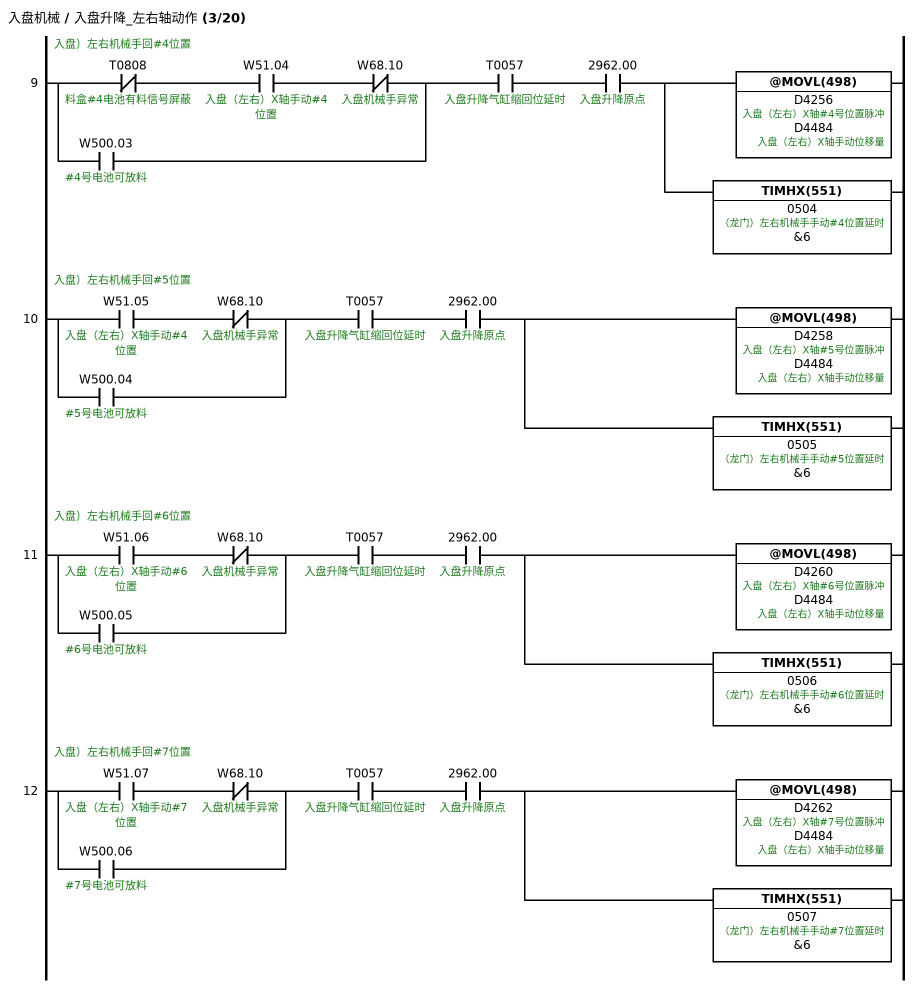
; [picture p192: 入盘机械 / 入盘升降_左右轴动作, rungs 9-12]
; rung 9: 入盘）左右机械手回#4位置
LDNOT T0808  ; 料盒#4电池有料信号屏蔽
AND W51.04  ; 入盘（左右）X轴手动#4位置
ANDNOT W68.10  ; 入盘机械手异常
OR W500.03  ; #4号电池可放料
AND T0057  ; 入盘升降气缸缩回位延时
AND 2962.00  ; 入盘升降原点
@MOVL(498) D4256 D4484  ; 入盘（左右）X轴#4号位置脉冲, 入盘（左右）X轴手动位移量
TIMHX(551) 0504 &6  ; （龙门）左右机械手手动#4位置延时
; rung 10: 入盘）左右机械手回#5位置
LD W51.05  ; 入盘（左右）X轴手动#4位置
ANDNOT W68.10  ; 入盘机械手异常
OR W500.04  ; #5号电池可放料
AND T0057  ; 入盘升降气缸缩回位延时
AND 2962.00  ; 入盘升降原点
@MOVL(498) D4258 D4484  ; 入盘（左右）X轴#5号位置脉冲, 入盘（左右）X轴手动位移量
TIMHX(551) 0505 &6  ; （龙门）左右机械手手动#5位置延时
; rung 11: 入盘）左右机械手回#6位置
LD W51.06  ; 入盘（左右）X轴手动#6位置
ANDNOT W68.10  ; 入盘机械手异常
OR W500.05  ; #6号电池可放料
AND T0057  ; 入盘升降气缸缩回位延时
AND 2962.00  ; 入盘升降原点
@MOVL(498) D4260 D4484  ; 入盘（左右）X轴#6号位置脉冲, 入盘（左右）X轴手动位移量
TIMHX(551) 0506 &6  ; （龙门）左右机械手手动#6位置延时
; rung 12: 入盘）左右机械手回#7位置
LD W51.07  ; 入盘（左右）X轴手动#7位置
ANDNOT W68.10  ; 入盘机械手异常
OR W500.06  ; #7号电池可放料
AND T0057  ; 入盘升降气缸缩回位延时
AND 2962.00  ; 入盘升降原点
@MOVL(498) D4262 D4484  ; 入盘（左右）X轴#7号位置脉冲, 入盘（左右）X轴手动位移量
TIMHX(551) 0507 &6  ; （龙门）左右机械手手动#7位置延时

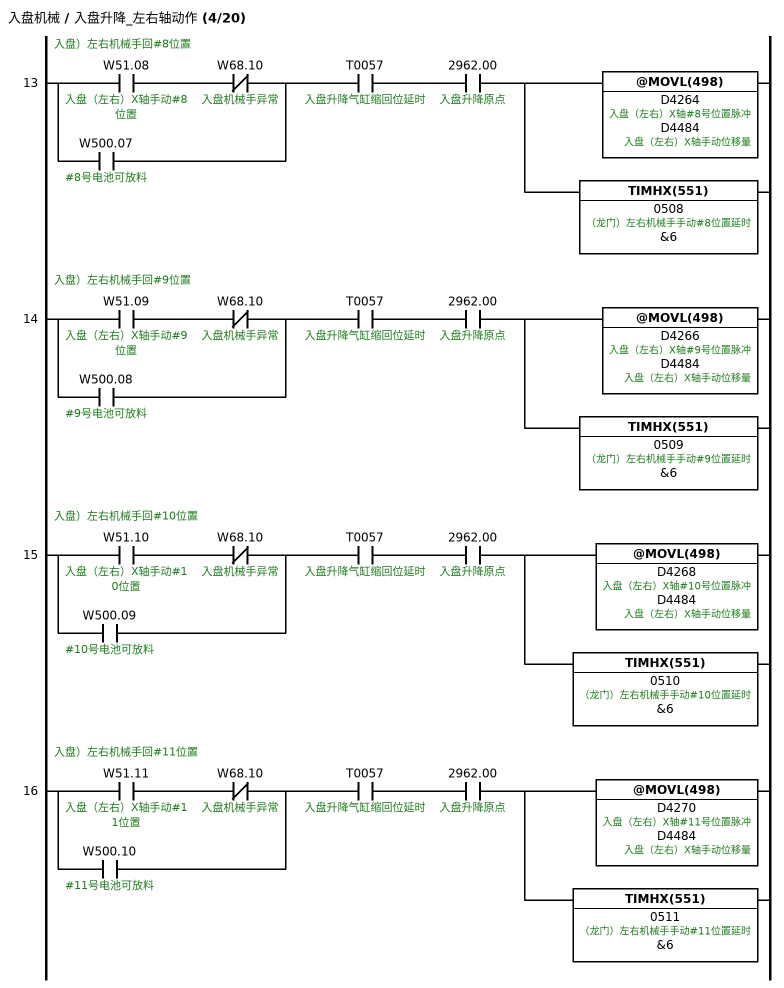
; rung 13: 入盘）左右机械手回#8位置
LD W51.08  ; 入盘（左右）X轴手动#8位置
ANDNOT W68.10  ; 入盘机械手异常
OR W500.07  ; #8号电池可放料
AND T0057  ; 入盘升降气缸缩回位延时
AND 2962.00  ; 入盘升降原点
@MOVL(498) D4264 D4484  ; 入盘（左右）X轴#8号位置脉冲, 入盘（左右）X轴手动位移量
TIMHX(551) 0508 &6  ; （龙门）左右机械手手动#8位置延时
; rung 14: 入盘）左右机械手回#9位置
LD W51.09  ; 入盘（左右）X轴手动#9位置
ANDNOT W68.10  ; 入盘机械手异常
OR W500.08  ; #9号电池可放料
AND T0057  ; 入盘升降气缸缩回位延时
AND 2962.00  ; 入盘升降原点
@MOVL(498) D4266 D4484  ; 入盘（左右）X轴#9号位置脉冲, 入盘（左右）X轴手动位移量
TIMHX(551) 0509 &6  ; （龙门）左右机械手手动#9位置延时
; rung 15: 入盘）左右机械手回#10位置
LD W51.10  ; 入盘（左右）X轴手动#10位置
ANDNOT W68.10  ; 入盘机械手异常
OR W500.09  ; #10号电池可放料
AND T0057  ; 入盘升降气缸缩回位延时
AND 2962.00  ; 入盘升降原点
@MOVL(498) D4268 D4484  ; 入盘（左右）X轴#10号位置脉冲, 入盘（左右）X轴手动位移量
TIMHX(551) 0510 &6  ; （龙门）左右机械手手动#10位置延时
; rung 16: 入盘）左右机械手回#11位置
LD W51.11  ; 入盘（左右）X轴手动#11位置
ANDNOT W68.10  ; 入盘机械手异常
OR W500.10  ; #11号电池可放料
AND T0057  ; 入盘升降气缸缩回位延时
AND 2962.00  ; 入盘升降原点
@MOVL(498) D4270 D4484  ; 入盘（左右）X轴#11号位置脉冲, 入盘（左右）X轴手动位移量
TIMHX(551) 0511 &6  ; （龙门）左右机械手手动#11位置延时

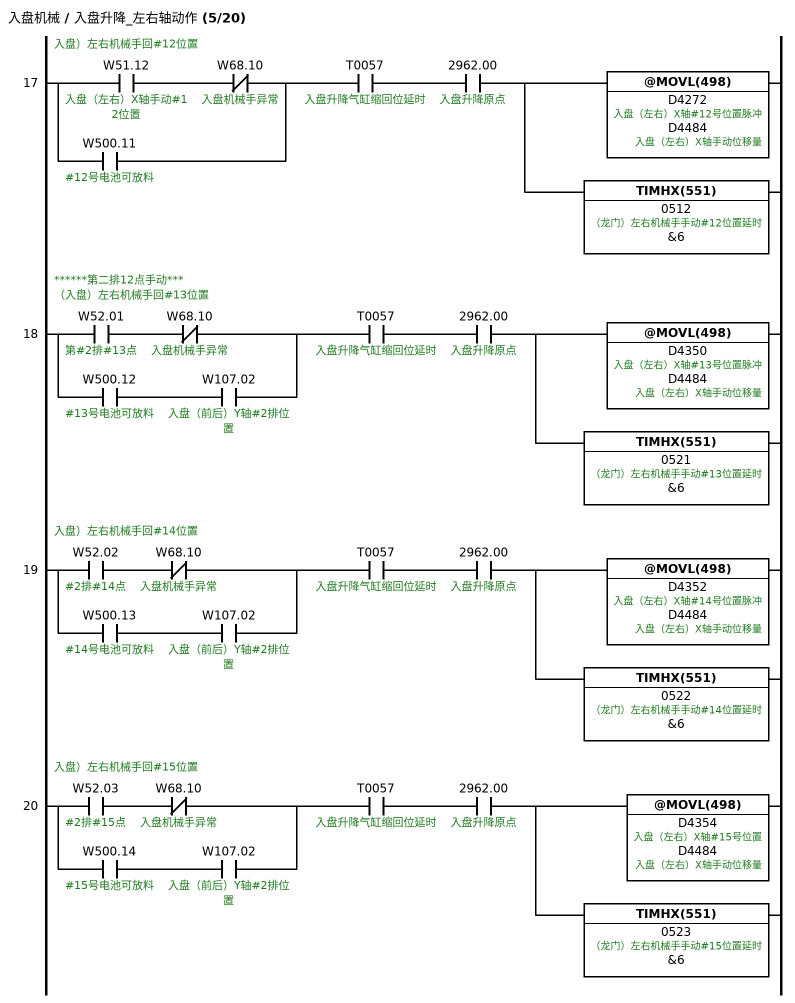
; rung 17: 入盘）左右机械手回#12位置
LD W51.12  ; 入盘（左右）X轴手动#12位置
ANDNOT W68.10  ; 入盘机械手异常
OR W500.11  ; #12号电池可放料
AND T0057  ; 入盘升降气缸缩回位延时
AND 2962.00  ; 入盘升降原点
@MOVL(498) D4272 D4484  ; 入盘（左右）X轴#12号位置脉冲, 入盘（左右）X轴手动位移量
TIMHX(551) 0512 &6  ; （龙门）左右机械手手动#12位置延时
; rung 18: ******第二排12点手动*** / （入盘）左右机械手回#13位置
LD W52.01  ; 第#2排#13点
ANDNOT W68.10  ; 入盘机械手异常
LD W500.12  ; #13号电池可放料
AND W107.02  ; 入盘（前后）Y轴#2排位置
ORLD
AND T0057  ; 入盘升降气缸缩回位延时
AND 2962.00  ; 入盘升降原点
@MOVL(498) D4350 D4484  ; 入盘（左右）X轴#13号位置脉冲, 入盘（左右）X轴手动位移量
TIMHX(551) 0521 &6  ; （龙门）左右机械手手动#13位置延时
; rung 19: 入盘）左右机械手回#14位置
LD W52.02  ; #2排#14点
ANDNOT W68.10  ; 入盘机械手异常
LD W500.13  ; #14号电池可放料
AND W107.02  ; 入盘（前后）Y轴#2排位置
ORLD
AND T0057  ; 入盘升降气缸缩回位延时
AND 2962.00  ; 入盘升降原点
@MOVL(498) D4352 D4484  ; 入盘（左右）X轴#14号位置脉冲, 入盘（左右）X轴手动位移量
TIMHX(551) 0522 &6  ; （龙门）左右机械手手动#14位置延时
; rung 20: 入盘）左右机械手回#15位置
LD W52.03  ; #2排#15点
ANDNOT W68.10  ; 入盘机械手异常
LD W500.14  ; #15号电池可放料
AND W107.02  ; 入盘（前后）Y轴#2排位置
ORLD
AND T0057  ; 入盘升降气缸缩回位延时
AND 2962.00  ; 入盘升降原点
@MOVL(498) D4354 D4484  ; 入盘（左右）X轴#15号位置, 入盘（左右）X轴手动位移量
TIMHX(551) 0523 &6  ; （龙门）左右机械手手动#15位置延时

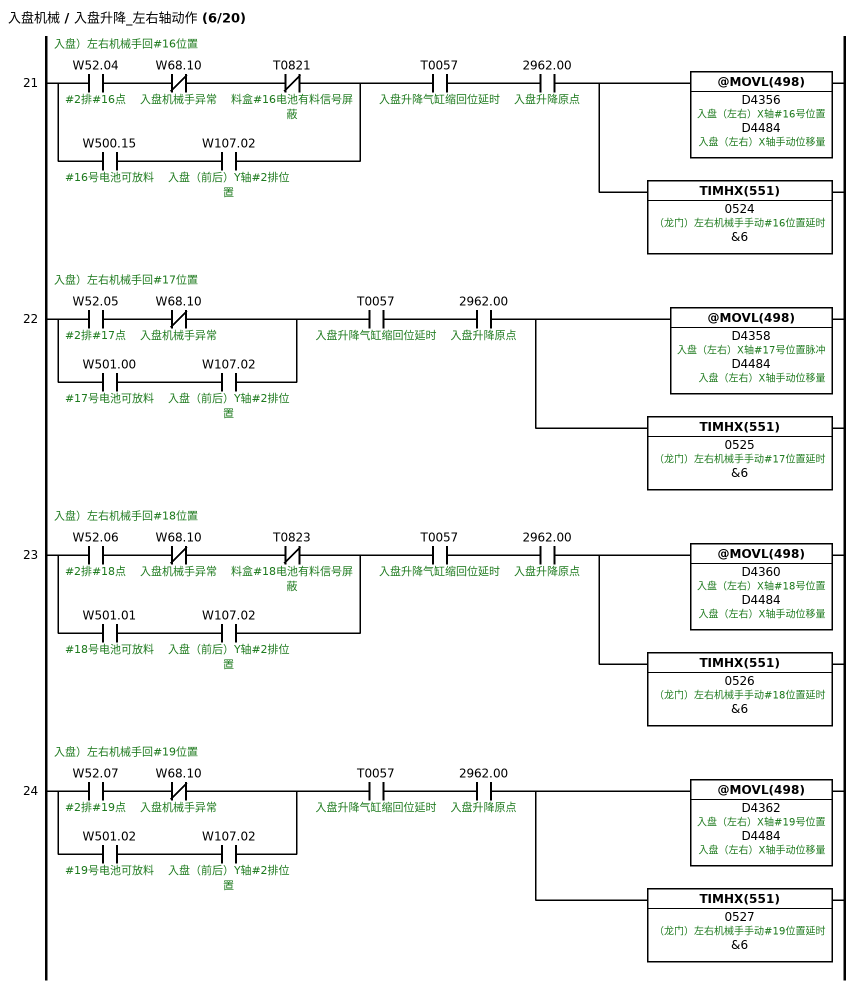
; rung 21: 入盘）左右机械手回#16位置
LD W52.04  ; #2排#16点
ANDNOT W68.10  ; 入盘机械手异常
ANDNOT T0821  ; 料盒#16电池有料信号屏蔽
LD W500.15  ; #16号电池可放料
AND W107.02  ; 入盘（前后）Y轴#2排位置
ORLD
AND T0057  ; 入盘升降气缸缩回位延时
AND 2962.00  ; 入盘升降原点
@MOVL(498) D4356 D4484  ; 入盘（左右）X轴#16号位置, 入盘（左右）X轴手动位移量
TIMHX(551) 0524 &6  ; （龙门）左右机械手手动#16位置延时
; rung 22: 入盘）左右机械手回#17位置
LD W52.05  ; #2排#17点
ANDNOT W68.10  ; 入盘机械手异常
LD W501.00  ; #17号电池可放料
AND W107.02  ; 入盘（前后）Y轴#2排位置
ORLD
AND T0057  ; 入盘升降气缸缩回位延时
AND 2962.00  ; 入盘升降原点
@MOVL(498) D4358 D4484  ; 入盘（左右）X轴#17号位置脉冲, 入盘（左右）X轴手动位移量
TIMHX(551) 0525 &6  ; （龙门）左右机械手手动#17位置延时
; rung 23: 入盘）左右机械手回#18位置
LD W52.06  ; #2排#18点
ANDNOT W68.10  ; 入盘机械手异常
ANDNOT T0823  ; 料盒#18电池有料信号屏蔽
LD W501.01  ; #18号电池可放料
AND W107.02  ; 入盘（前后）Y轴#2排位置
ORLD
AND T0057  ; 入盘升降气缸缩回位延时
AND 2962.00  ; 入盘升降原点
@MOVL(498) D4360 D4484  ; 入盘（左右）X轴#18号位置, 入盘（左右）X轴手动位移量
TIMHX(551) 0526 &6  ; （龙门）左右机械手手动#18位置延时
; rung 24: 入盘）左右机械手回#19位置
LD W52.07  ; #2排#19点
ANDNOT W68.10  ; 入盘机械手异常
LD W501.02  ; #19号电池可放料
AND W107.02  ; 入盘（前后）Y轴#2排位置
ORLD
AND T0057  ; 入盘升降气缸缩回位延时
AND 2962.00  ; 入盘升降原点
@MOVL(498) D4362 D4484  ; 入盘（左右）X轴#19号位置, 入盘（左右）X轴手动位移量
TIMHX(551) 0527 &6  ; （龙门）左右机械手手动#19位置延时

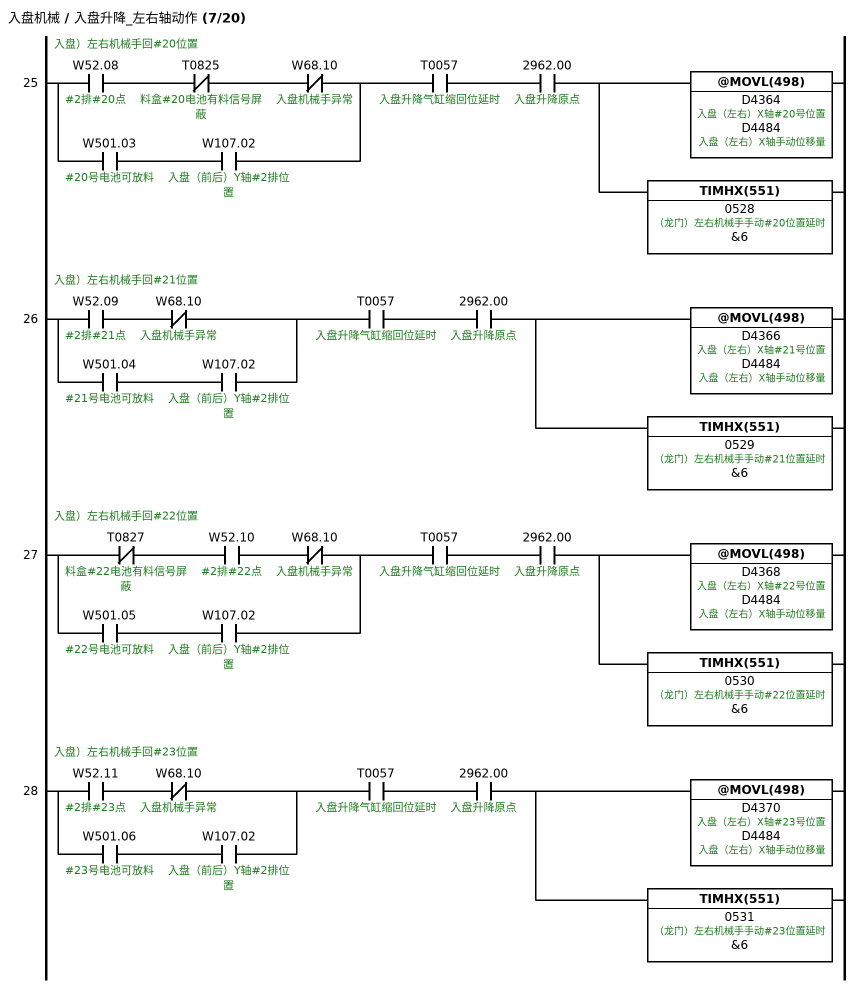
; rung 25: 入盘）左右机械手回#20位置
LD W52.08  ; #2排#20点
ANDNOT T0825  ; 料盒#20电池有料信号屏蔽
ANDNOT W68.10  ; 入盘机械手异常
LD W501.03  ; #20号电池可放料
AND W107.02  ; 入盘（前后）Y轴#2排位置
ORLD
AND T0057  ; 入盘升降气缸缩回位延时
AND 2962.00  ; 入盘升降原点
@MOVL(498) D4364 D4484  ; 入盘（左右）X轴#20号位置, 入盘（左右）X轴手动位移量
TIMHX(551) 0528 &6  ; （龙门）左右机械手手动#20位置延时
; rung 26: 入盘）左右机械手回#21位置
LD W52.09  ; #2排#21点
ANDNOT W68.10  ; 入盘机械手异常
LD W501.04  ; #21号电池可放料
AND W107.02  ; 入盘（前后）Y轴#2排位置
ORLD
AND T0057  ; 入盘升降气缸缩回位延时
AND 2962.00  ; 入盘升降原点
@MOVL(498) D4366 D4484  ; 入盘（左右）X轴#21号位置, 入盘（左右）X轴手动位移量
TIMHX(551) 0529 &6  ; （龙门）左右机械手手动#21位置延时
; rung 27: 入盘）左右机械手回#22位置
LDNOT T0827  ; 料盒#22电池有料信号屏蔽
AND W52.10  ; #2排#22点
ANDNOT W68.10  ; 入盘机械手异常
LD W501.05  ; #22号电池可放料
AND W107.02  ; 入盘（前后）Y轴#2排位置
ORLD
AND T0057  ; 入盘升降气缸缩回位延时
AND 2962.00  ; 入盘升降原点
@MOVL(498) D4368 D4484  ; 入盘（左右）X轴#22号位置, 入盘（左右）X轴手动位移量
TIMHX(551) 0530 &6  ; （龙门）左右机械手手动#22位置延时
; rung 28: 入盘）左右机械手回#23位置
LD W52.11  ; #2排#23点
ANDNOT W68.10  ; 入盘机械手异常
LD W501.06  ; #23号电池可放料
AND W107.02  ; 入盘（前后）Y轴#2排位置
ORLD
AND T0057  ; 入盘升降气缸缩回位延时
AND 2962.00  ; 入盘升降原点
@MOVL(498) D4370 D4484  ; 入盘（左右）X轴#23号位置, 入盘（左右）X轴手动位移量
TIMHX(551) 0531 &6  ; （龙门）左右机械手手动#23位置延时

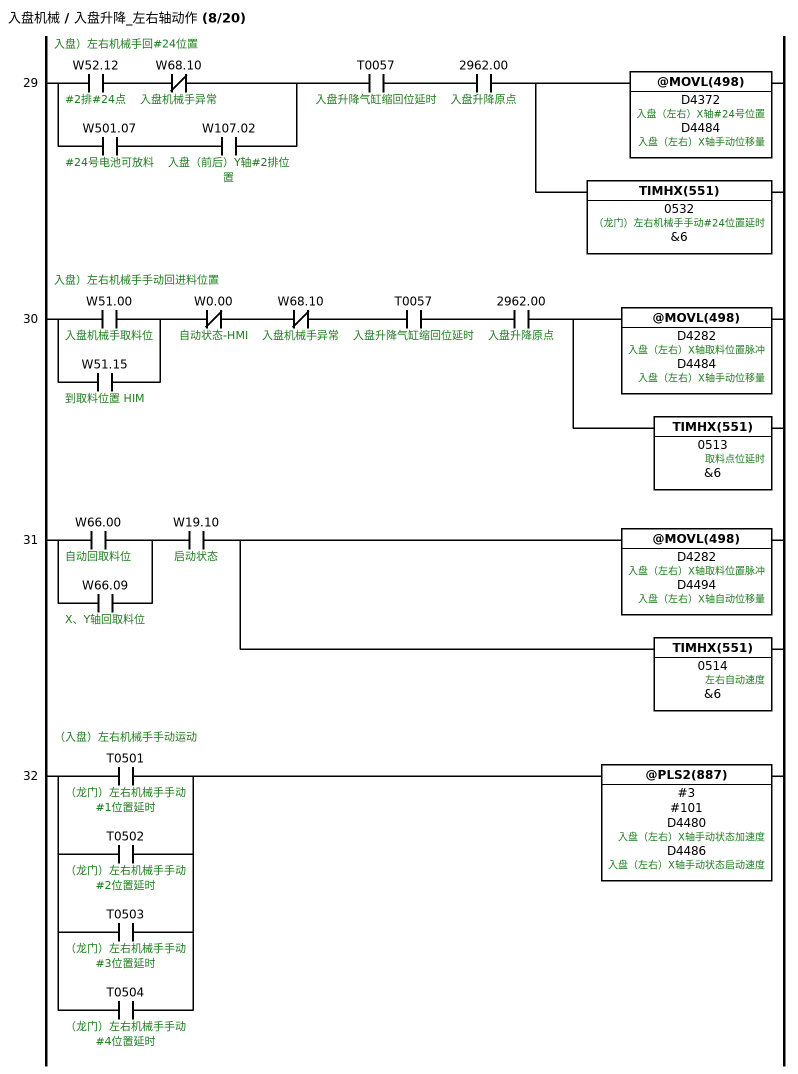
; rung 29: 入盘）左右机械手回#24位置
LD W52.12  ; #2排#24点
ANDNOT W68.10  ; 入盘机械手异常
LD W501.07  ; #24号电池可放料
AND W107.02  ; 入盘（前后）Y轴#2排位置
ORLD
AND T0057  ; 入盘升降气缸缩回位延时
AND 2962.00  ; 入盘升降原点
@MOVL(498) D4372 D4484  ; 入盘（左右）X轴#24号位置, 入盘（左右）X轴手动位移量
TIMHX(551) 0532 &6  ; （龙门）左右机械手手动#24位置延时
; rung 30: 入盘）左右机械手手动回进料位置
LD W51.00  ; 入盘机械手取料位
OR W51.15  ; 到取料位置 HIM
ANDNOT W0.00  ; 自动状态-HMI
ANDNOT W68.10  ; 入盘机械手异常
AND T0057  ; 入盘升降气缸缩回位延时
AND 2962.00  ; 入盘升降原点
@MOVL(498) D4282 D4484  ; 入盘（左右）X轴取料位置脉冲, 入盘（左右）X轴手动位移量
TIMHX(551) 0513 &6  ; 取料点位延时
; rung 31
LD W66.00  ; 自动回取料位
OR W66.09  ; X、Y轴回取料位
AND W19.10  ; 启动状态
@MOVL(498) D4282 D4494  ; 入盘（左右）X轴取料位置脉冲, 入盘（左右）X轴自动位移量
TIMHX(551) 0514 &6  ; 左右自动速度
; rung 32: （入盘）左右机械手手动运动
LD T0501  ; （龙门）左右机械手手动#1位置延时
OR T0502  ; （龙门）左右机械手手动#2位置延时
OR T0503  ; （龙门）左右机械手手动#3位置延时
OR T0504  ; （龙门）左右机械手手动#4位置延时
@PLS2(887) #3 #101 D4480 D4486  ; 入盘（左右）X轴手动状态加速度, 入盘（左右）X轴手动状态启动速度

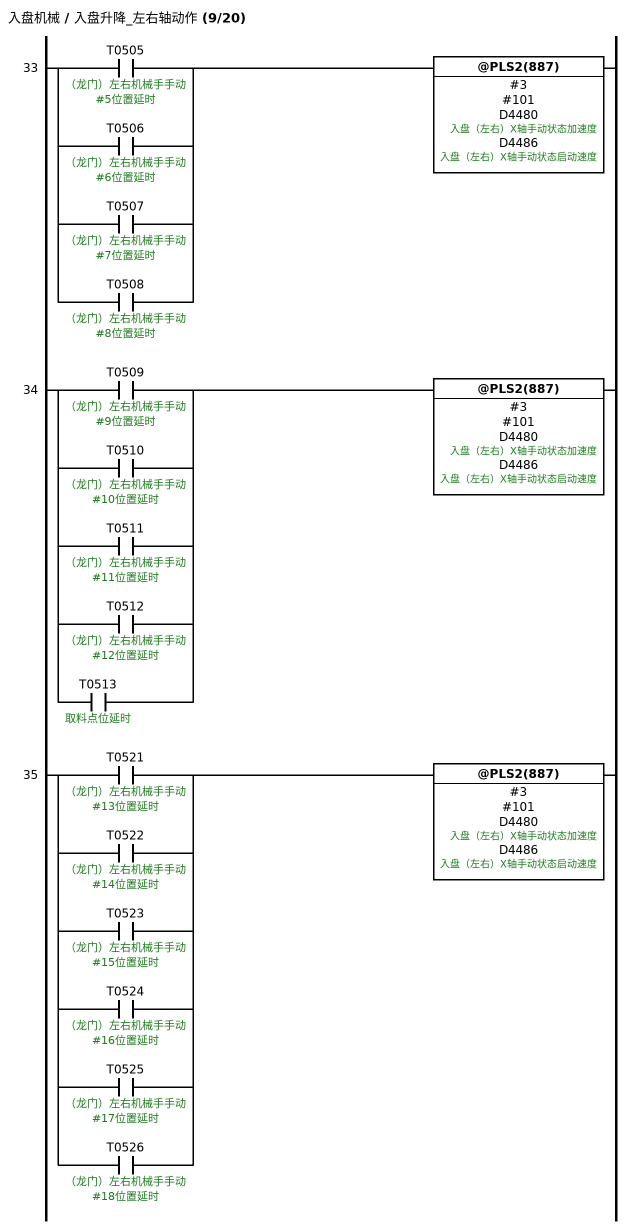
; rung 33
LD T0505  ; （龙门）左右机械手手动#5位置延时
OR T0506  ; （龙门）左右机械手手动#6位置延时
OR T0507  ; （龙门）左右机械手手动#7位置延时
OR T0508  ; （龙门）左右机械手手动#8位置延时
@PLS2(887) #3 #101 D4480 D4486  ; 入盘（左右）X轴手动状态加速度, 入盘（左右）X轴手动状态启动速度
; rung 34
LD T0509  ; （龙门）左右机械手手动#9位置延时
OR T0510  ; （龙门）左右机械手手动#10位置延时
OR T0511  ; （龙门）左右机械手手动#11位置延时
OR T0512  ; （龙门）左右机械手手动#12位置延时
OR T0513  ; 取料点位延时
@PLS2(887) #3 #101 D4480 D4486  ; 入盘（左右）X轴手动状态加速度, 入盘（左右）X轴手动状态启动速度
; rung 35
LD T0521  ; （龙门）左右机械手手动#13位置延时
OR T0522  ; （龙门）左右机械手手动#14位置延时
OR T0523  ; （龙门）左右机械手手动#15位置延时
OR T0524  ; （龙门）左右机械手手动#16位置延时
OR T0525  ; （龙门）左右机械手手动#17位置延时
OR T0526  ; （龙门）左右机械手手动#18位置延时
@PLS2(887) #3 #101 D4480 D4486  ; 入盘（左右）X轴手动状态加速度, 入盘（左右）X轴手动状态启动速度

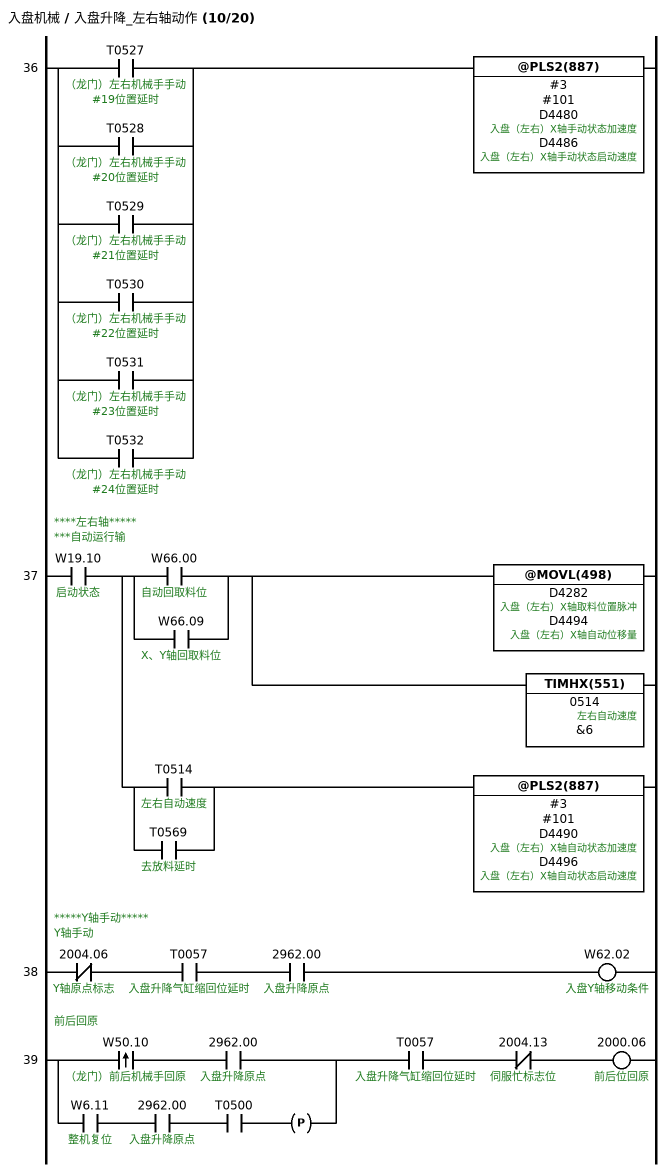
; rung 36
LD T0527  ; （龙门）左右机械手手动#19位置延时
OR T0528  ; （龙门）左右机械手手动#20位置延时
OR T0529  ; （龙门）左右机械手手动#21位置延时
OR T0530  ; （龙门）左右机械手手动#22位置延时
OR T0531  ; （龙门）左右机械手手动#23位置延时
OR T0532  ; （龙门）左右机械手手动#24位置延时
@PLS2(887) #3 #101 D4480 D4486  ; 入盘（左右）X轴手动状态加速度, 入盘（左右）X轴手动状态启动速度
; rung 37: ****左右轴***** / ***自动运行输
LD W19.10  ; 启动状态
OUT TR0
LD W66.00  ; 自动回取料位
OR W66.09  ; X、Y轴回取料位
ANDLD
@MOVL(498) D4282 D4494  ; 入盘（左右）X轴取料位置脉冲, 入盘（左右）X轴自动位移量
TIMHX(551) 0514 &6  ; 左右自动速度
LD TR0
LD T0514  ; 左右自动速度
OR T0569  ; 去放料延时
ANDLD
@PLS2(887) #3 #101 D4490 D4496  ; 入盘（左右）X轴自动状态加速度, 入盘（左右）X轴自动状态启动速度
; rung 38: *****Y轴手动***** / Y轴手动
LDNOT 2004.06  ; Y轴原点标志
AND T0057  ; 入盘升降气缸缩回位延时
AND 2962.00  ; 入盘升降原点
OUT W62.02  ; 入盘Y轴移动条件
; rung 39: 前后回原
@LD W50.10  ; （龙门）前后机械手回原
AND 2962.00  ; 入盘升降原点
LD W6.11  ; 整机复位
AND 2962.00  ; 入盘升降原点
AND T0500
UP(521)
ORLD
AND T0057  ; 入盘升降气缸缩回位延时
ANDNOT 2004.13  ; 伺服忙标志位
OUT 2000.06  ; 前后位回原

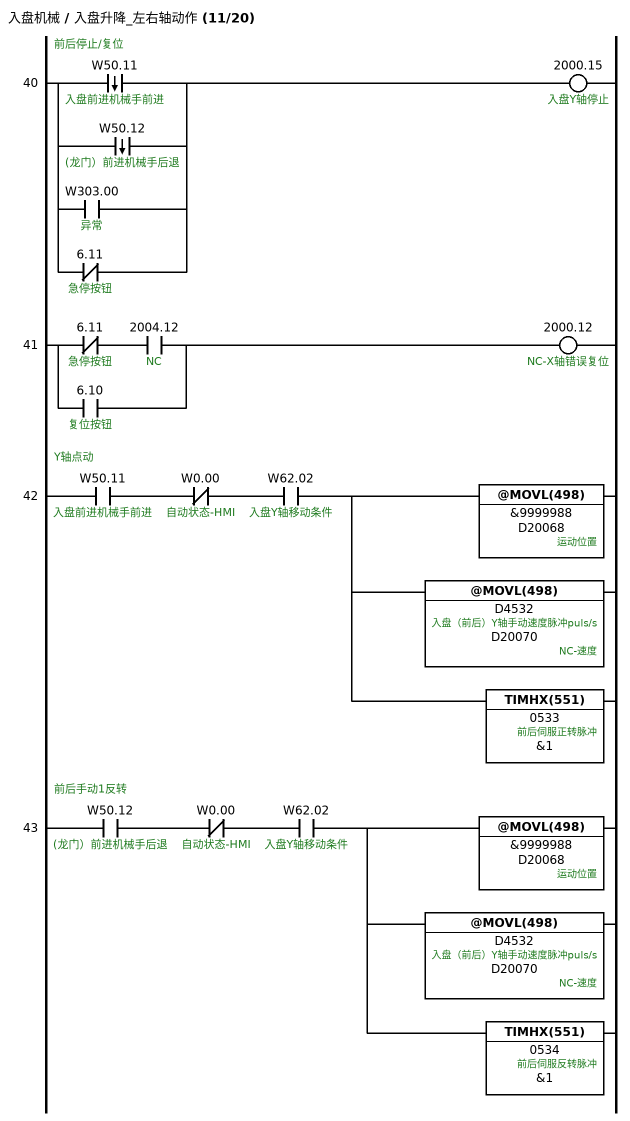
; rung 40: 前后停止/复位
%LD W50.11  ; 入盘前进机械手前进
%OR W50.12  ; (龙门）前进机械手后退
OR W303.00  ; 异常
ORNOT 6.11  ; 急停按钮
OUT 2000.15  ; 入盘Y轴停止
; rung 41
LDNOT 6.11  ; 急停按钮
AND 2004.12  ; NC
OR 6.10  ; 复位按钮
OUT 2000.12  ; NC-X轴错误复位
; rung 42: Y轴点动
LD W50.11  ; 入盘前进机械手前进
ANDNOT W0.00  ; 自动状态-HMI
AND W62.02  ; 入盘Y轴移动条件
@MOVL(498) &9999988 D20068  ; 运动位置
@MOVL(498) D4532 D20070  ; 入盘（前后）Y轴手动速度脉冲puls/s, NC-速度
TIMHX(551) 0533 &1  ; 前后伺服正转脉冲
; rung 43: 前后手动1反转
LD W50.12  ; (龙门）前进机械手后退
ANDNOT W0.00  ; 自动状态-HMI
AND W62.02  ; 入盘Y轴移动条件
@MOVL(498) &9999988 D20068  ; 运动位置
@MOVL(498) D4532 D20070  ; 入盘（前后）Y轴手动速度脉冲puls/s, NC-速度
TIMHX(551) 0534 &1  ; 前后伺服反转脉冲

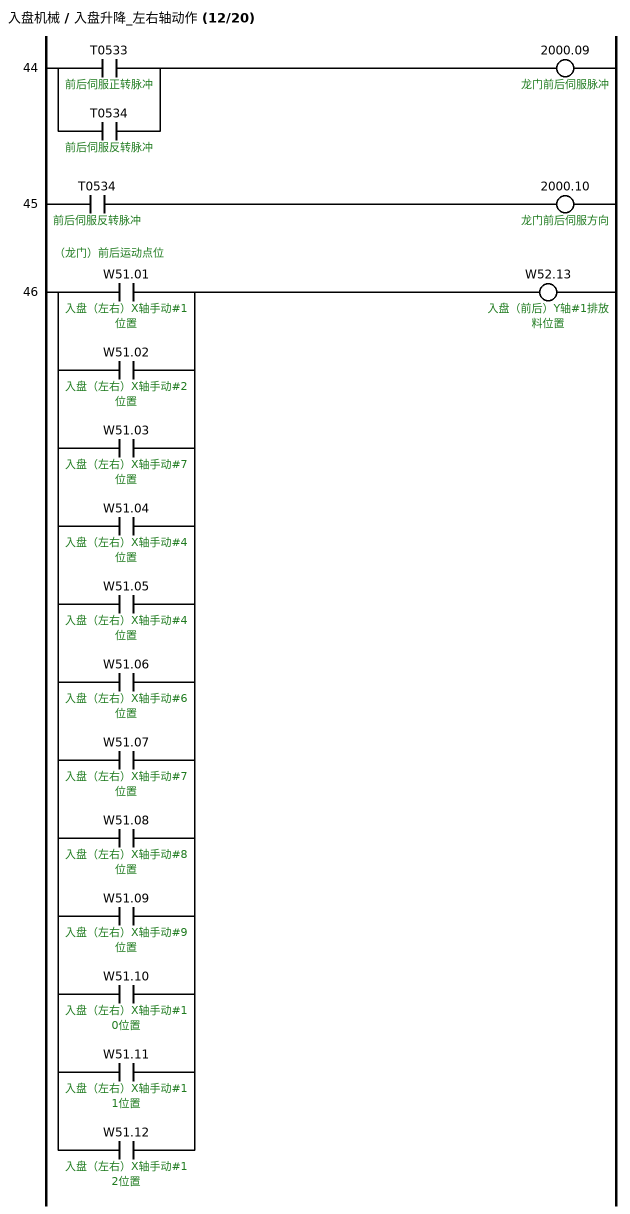
; rung 44
LD T0533  ; 前后伺服正转脉冲
OR T0534  ; 前后伺服反转脉冲
OUT 2000.09  ; 龙门前后伺服脉冲
; rung 45
LD T0534  ; 前后伺服反转脉冲
OUT 2000.10  ; 龙门前后伺服方向
; rung 46: （龙门）前后运动点位
LD W51.01  ; 入盘（左右）X轴手动#1位置
OR W51.02  ; 入盘（左右）X轴手动#2位置
OR W51.03  ; 入盘（左右）X轴手动#7位置
OR W51.04  ; 入盘（左右）X轴手动#4位置
OR W51.05  ; 入盘（左右）X轴手动#4位置
OR W51.06  ; 入盘（左右）X轴手动#6位置
OR W51.07  ; 入盘（左右）X轴手动#7位置
OR W51.08  ; 入盘（左右）X轴手动#8位置
OR W51.09  ; 入盘（左右）X轴手动#9位置
OR W51.10  ; 入盘（左右）X轴手动#10位置
OR W51.11  ; 入盘（左右）X轴手动#11位置
OR W51.12  ; 入盘（左右）X轴手动#12位置
OUT W52.13  ; 入盘（前后）Y轴#1排放料位置

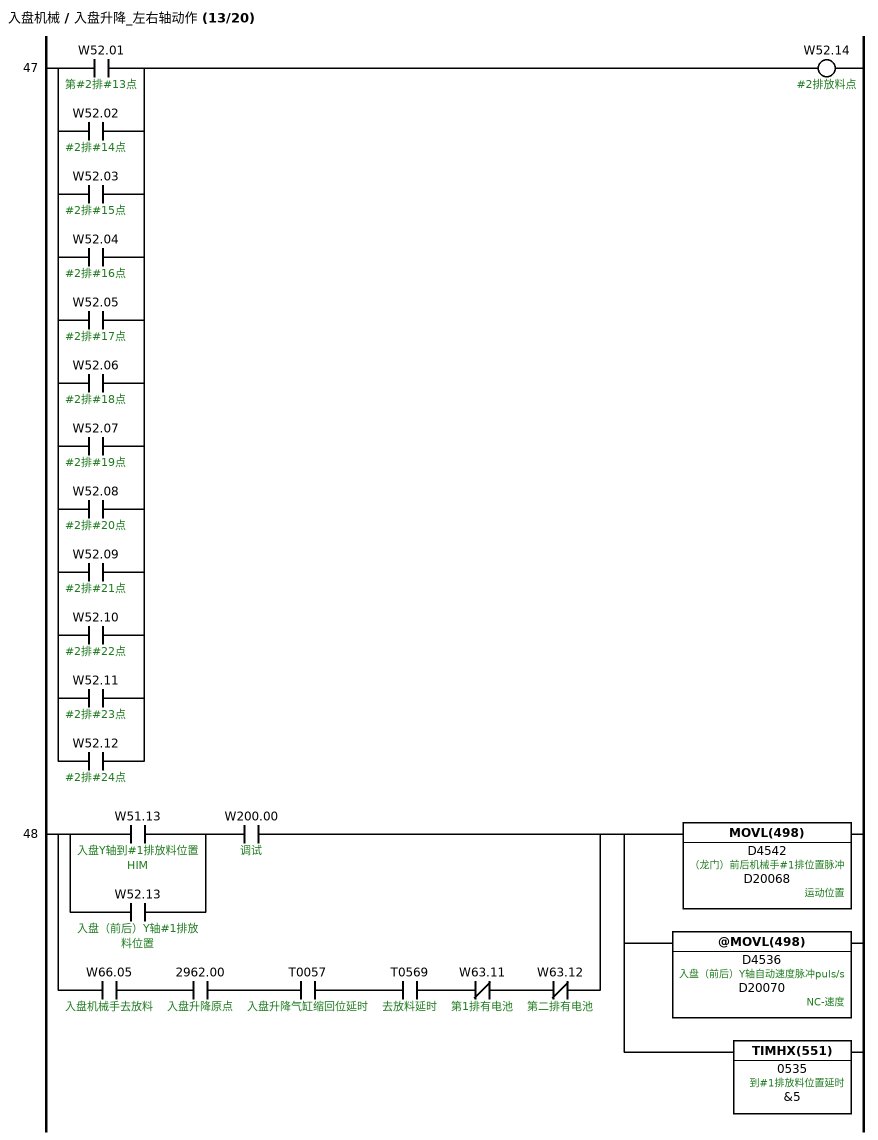
; rung 47
LD W52.01  ; 第#2排#13点
OR W52.02  ; #2排#14点
OR W52.03  ; #2排#15点
OR W52.04  ; #2排#16点
OR W52.05  ; #2排#17点
OR W52.06  ; #2排#18点
OR W52.07  ; #2排#19点
OR W52.08  ; #2排#20点
OR W52.09  ; #2排#21点
OR W52.10  ; #2排#22点
OR W52.11  ; #2排#23点
OR W52.12  ; #2排#24点
OUT W52.14  ; #2排放料点
; rung 48
LD W51.13  ; 入盘Y轴到#1排放料位置  HIM
OR W52.13  ; 入盘（前后）Y轴#1排放料位置
AND W200.00  ; 调试
LD W66.05  ; 入盘机械手去放料
AND 2962.00  ; 入盘升降原点
AND T0057  ; 入盘升降气缸缩回位延时
AND T0569  ; 去放料延时
ANDNOT W63.11  ; 第1排有电池
ANDNOT W63.12  ; 第二排有电池
ORLD
MOVL(498) D4542 D20068  ; （龙门）前后机械手#1排位置脉冲, 运动位置
@MOVL(498) D4536 D20070  ; 入盘（前后）Y轴自动速度脉冲puls/s, NC-速度
TIMHX(551) 0535 &5  ; 到#1排放料位置延时

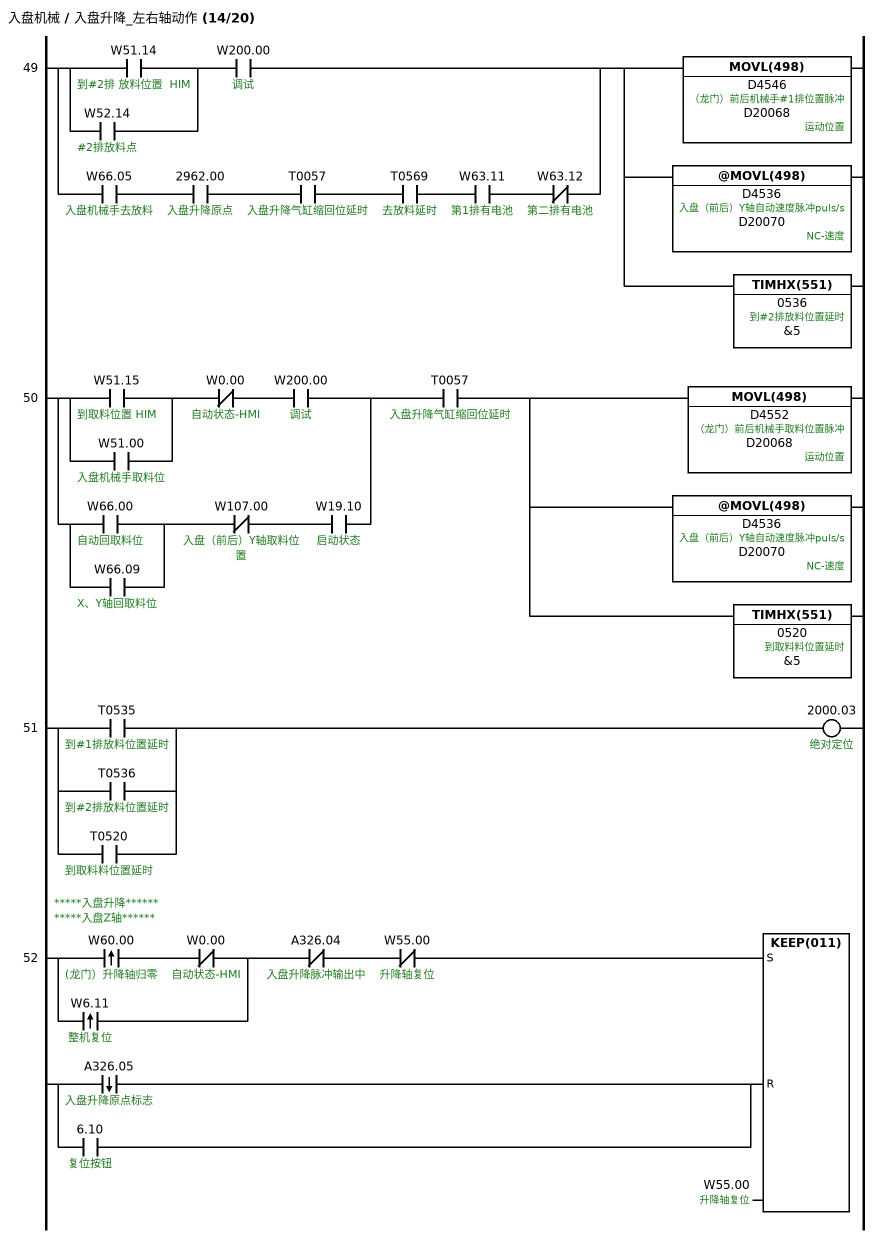
; rung 49
LD W51.14  ; 到#2排 放料位置  HIM
OR W52.14  ; #2排放料点
AND W200.00  ; 调试
LD W66.05  ; 入盘机械手去放料
AND 2962.00  ; 入盘升降原点
AND T0057  ; 入盘升降气缸缩回位延时
AND T0569  ; 去放料延时
AND W63.11  ; 第1排有电池
ANDNOT W63.12  ; 第二排有电池
ORLD
MOVL(498) D4546 D20068  ; （龙门）前后机械手#1排位置脉冲, 运动位置
@MOVL(498) D4536 D20070  ; 入盘（前后）Y轴自动速度脉冲puls/s, NC-速度
TIMHX(551) 0536 &5  ; 到#2排放料位置延时
; rung 50
LD W51.15  ; 到取料位置 HIM
OR W51.00  ; 入盘机械手取料位
ANDNOT W0.00  ; 自动状态-HMI
AND W200.00  ; 调试
LD W66.00  ; 自动回取料位
OR W66.09  ; X、Y轴回取料位
ANDNOT W107.00  ; 入盘（前后）Y轴取料位置
AND W19.10  ; 启动状态
ORLD
AND T0057  ; 入盘升降气缸缩回位延时
MOVL(498) D4552 D20068  ; （龙门）前后机械手取料位置脉冲, 运动位置
@MOVL(498) D4536 D20070  ; 入盘（前后）Y轴自动速度脉冲puls/s, NC-速度
TIMHX(551) 0520 &5  ; 到取料料位置延时
; rung 51
LD T0535  ; 到#1排放料位置延时
OR T0536  ; 到#2排放料位置延时
OR T0520  ; 到取料料位置延时
OUT 2000.03  ; 绝对定位
; rung 52: *****入盘升降****** / *****入盘Z轴******
@LD W60.00  ; (龙门）升降轴归零
ANDNOT W0.00  ; 自动状态-HMI
@OR W6.11  ; 整机复位
ANDNOT A326.04  ; 入盘升降脉冲输出中
ANDNOT W55.00  ; 升降轴复位
%LD A326.05  ; 入盘升降原点标志
OR 6.10  ; 复位按钮
KEEP(011) W55.00  ; 升降轴复位

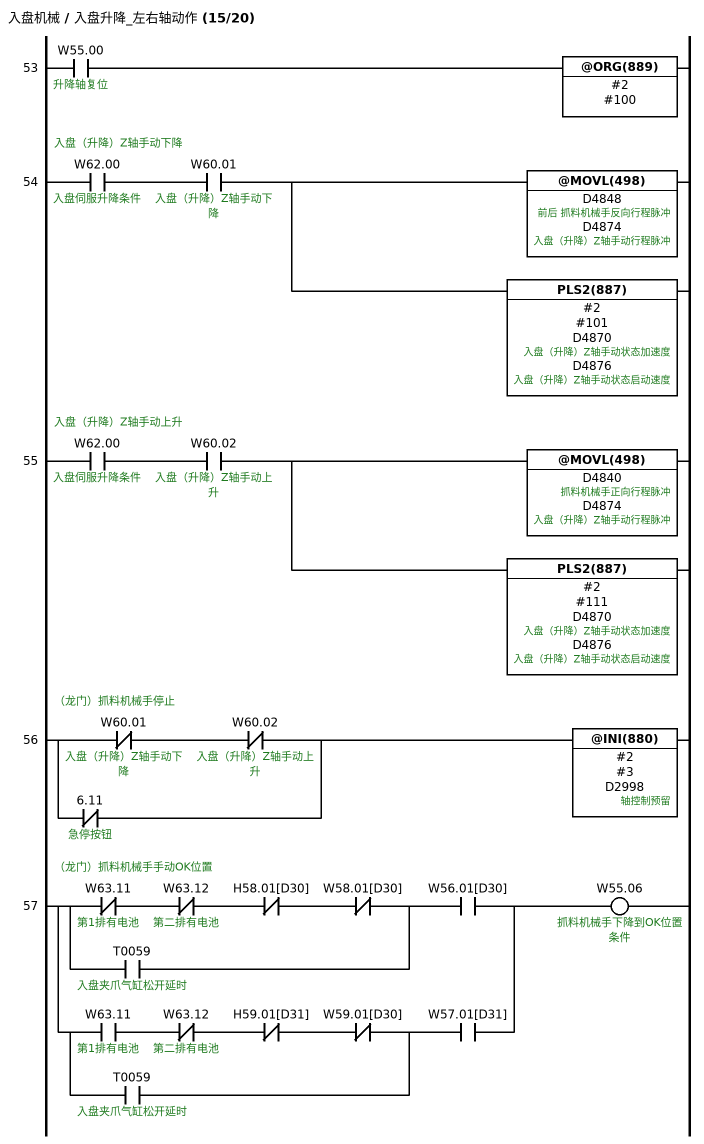
; rung 53
LD W55.00  ; 升降轴复位
@ORG(889) #2 #100
; rung 54: 入盘（升降）Z轴手动下降
LD W62.00  ; 入盘伺服升降条件
AND W60.01  ; 入盘（升降）Z轴手动下降
@MOVL(498) D4848 D4874  ; 前后 抓料机械手反向行程脉冲, 入盘（升降）Z轴手动行程脉冲
PLS2(887) #2 #101 D4870 D4876  ; 入盘（升降）Z轴手动状态加速度, 入盘（升降）Z轴手动状态启动速度
; rung 55: 入盘（升降）Z轴手动上升
LD W62.00  ; 入盘伺服升降条件
AND W60.02  ; 入盘（升降）Z轴手动上升
@MOVL(498) D4840 D4874  ; 抓料机械手正向行程脉冲, 入盘（升降）Z轴手动行程脉冲
PLS2(887) #2 #111 D4870 D4876  ; 入盘（升降）Z轴手动状态加速度, 入盘（升降）Z轴手动状态启动速度
; rung 56: （龙门）抓料机械手停止
LDNOT W60.01  ; 入盘（升降）Z轴手动下降
ANDNOT W60.02  ; 入盘（升降）Z轴手动上升
ORNOT 6.11  ; 急停按钮
@INI(880) #2 #3 D2998  ; 轴控制预留
; rung 57: （龙门）抓料机械手手动OK位置
LDNOT W63.11  ; 第1排有电池
ANDNOT W63.12  ; 第二排有电池
ANDNOT H58.01[D30]
ANDNOT W58.01[D30]
OR T0059  ; 入盘夹爪气缸松开延时
AND W56.01[D30]
LD W63.11  ; 第1排有电池
ANDNOT W63.12  ; 第二排有电池
ANDNOT H59.01[D31]
ANDNOT W59.01[D30]
OR T0059  ; 入盘夹爪气缸松开延时
AND W57.01[D31]
ORLD
OUT W55.06  ; 抓料机械手下降到OK位置条件

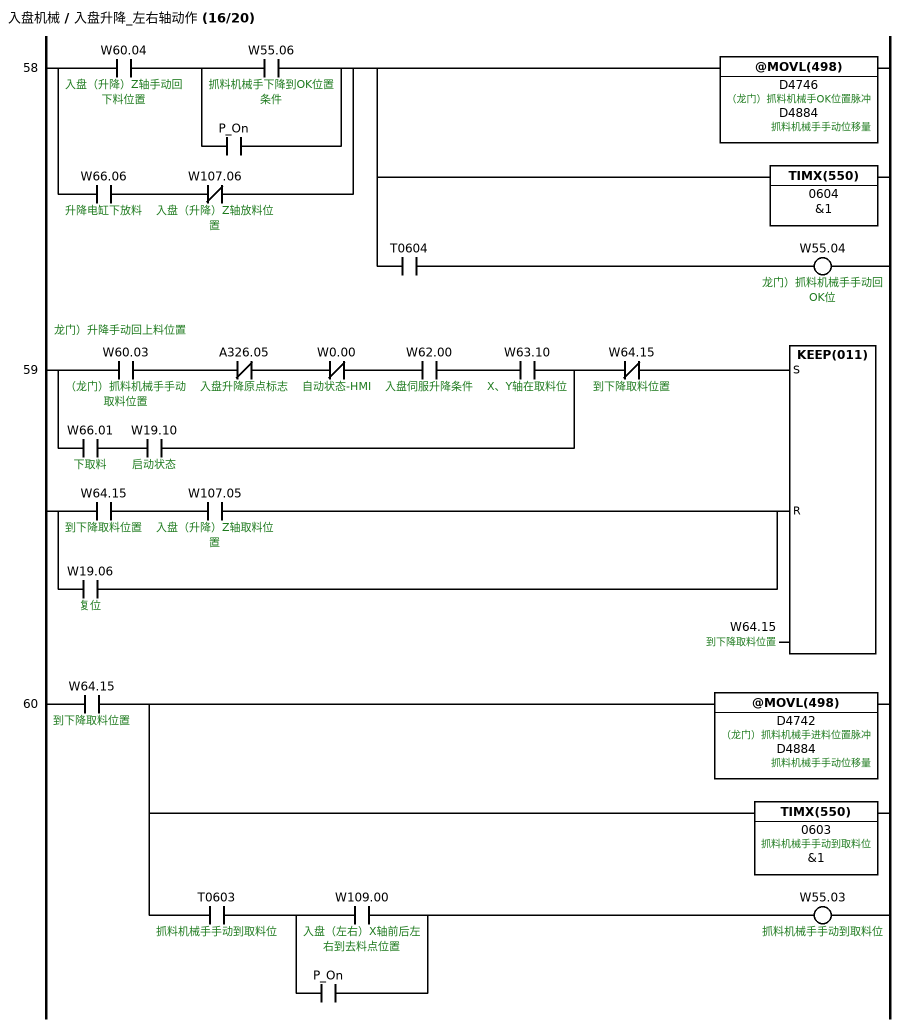
; rung 58
LD W60.04  ; 入盘（升降）Z轴手动回下料位置
LD W55.06  ; 抓料机械手下降到OK位置条件
OR P_On
ANDLD
LD W66.06  ; 升降电缸下放料
ANDNOT W107.06  ; 入盘（升降）Z轴放料位置
ORLD
@MOVL(498) D4746 D4884  ; （龙门）抓料机械手OK位置脉冲, 抓料机械手手动位移量
TIMX(550) 0604 &1
AND T0604
OUT W55.04  ; 龙门）抓料机械手手动回OK位
; rung 59: 龙门）升降手动回上料位置
LD W60.03  ; （龙门）抓料机械手手动取料位置
ANDNOT A326.05  ; 入盘升降原点标志
ANDNOT W0.00  ; 自动状态-HMI
AND W62.00  ; 入盘伺服升降条件
AND W63.10  ; X、Y轴在取料位
LD W66.01  ; 下取料
AND W19.10  ; 启动状态
ORLD
ANDNOT W64.15  ; 到下降取料位置
LD W64.15  ; 到下降取料位置
AND W107.05  ; 入盘（升降）Z轴取料位置
OR W19.06  ; 复位
KEEP(011) W64.15  ; 到下降取料位置
; rung 60
LD W64.15  ; 到下降取料位置
@MOVL(498) D4742 D4884  ; （龙门）抓料机械手进料位置脉冲, 抓料机械手手动位移量
TIMX(550) 0603 &1  ; 抓料机械手手动到取料位
AND T0603  ; 抓料机械手手动到取料位
LD W109.00  ; 入盘（左右）X轴前后左右到去料点位置
OR P_On
ANDLD
OUT W55.03  ; 抓料机械手手动到取料位

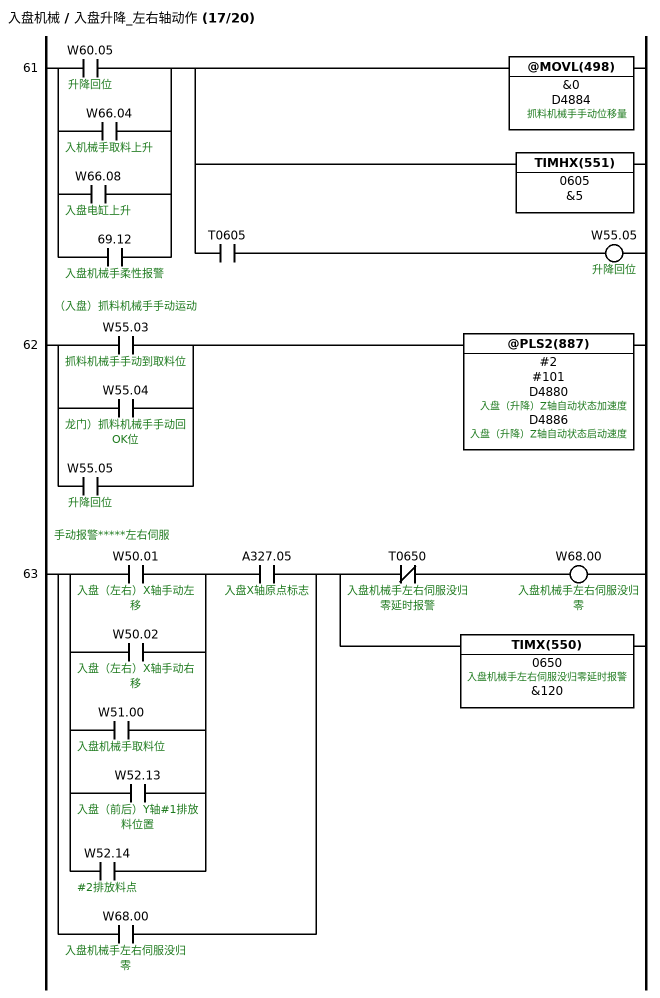
; rung 61
LD W60.05  ; 升降回位
OR W66.04  ; 入机械手取料上升
OR W66.08  ; 入盘电缸上升
OR 69.12  ; 入盘机械手柔性报警
@MOVL(498) &0 D4884  ; 抓料机械手手动位移量
TIMHX(551) 0605 &5
AND T0605
OUT W55.05  ; 升降回位
; rung 62: （入盘）抓料机械手手动运动
LD W55.03  ; 抓料机械手手动到取料位
OR W55.04  ; 龙门）抓料机械手手动回OK位
OR W55.05  ; 升降回位
@PLS2(887) #2 #101 D4880 D4886  ; 入盘（升降）Z轴自动状态加速度, 入盘（升降）Z轴自动状态启动速度
; rung 63: 手动报警*****左右伺服
LD W50.01  ; 入盘（左右）X轴手动左移
OR W50.02  ; 入盘（左右）X轴手动右移
OR W51.00  ; 入盘机械手取料位
OR W52.13  ; 入盘（前后）Y轴#1排放料位置
OR W52.14  ; #2排放料点
AND A327.05  ; 入盘X轴原点标志
OR W68.00  ; 入盘机械手左右伺服没归零
OUT TR0
ANDNOT T0650  ; 入盘机械手左右伺服没归零延时报警
OUT W68.00  ; 入盘机械手左右伺服没归零
LD TR0
TIMX(550) 0650 &120  ; 入盘机械手左右伺服没归零延时报警

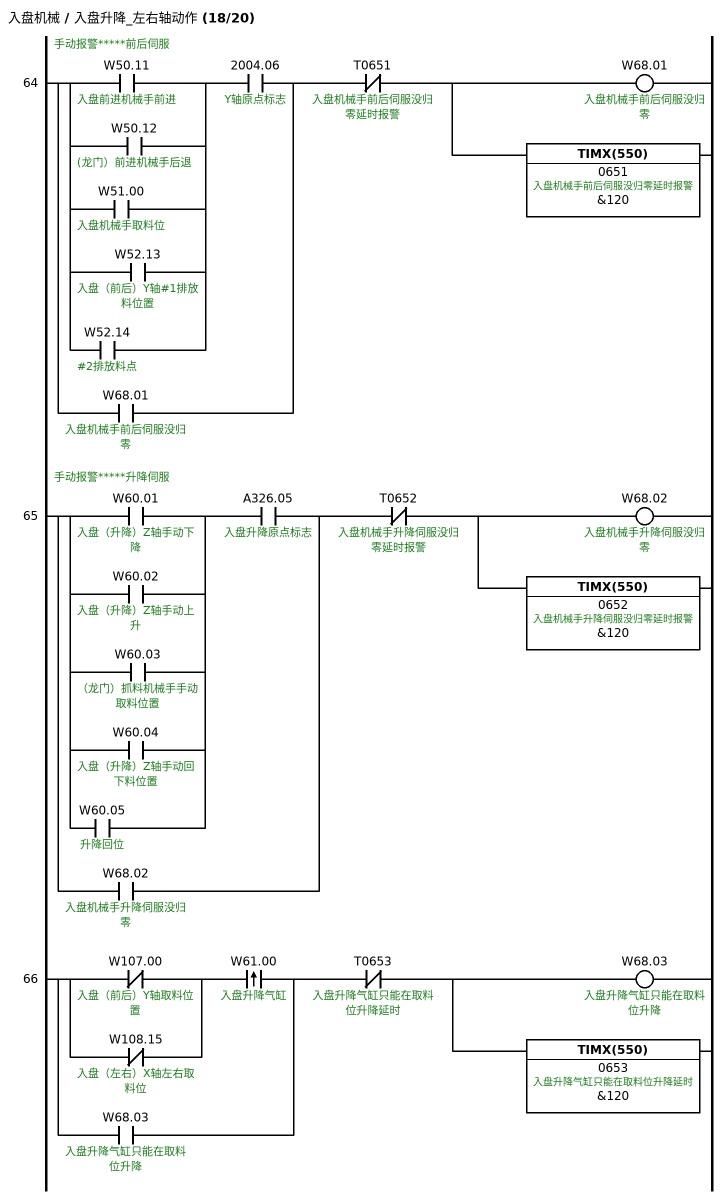
; rung 64: 手动报警*****前后伺服
LD W50.11  ; 入盘前进机械手前进
OR W50.12  ; (龙门）前进机械手后退
OR W51.00  ; 入盘机械手取料位
OR W52.13  ; 入盘（前后）Y轴#1排放料位置
OR W52.14  ; #2排放料点
AND 2004.06  ; Y轴原点标志
OR W68.01  ; 入盘机械手前后伺服没归零
ANDNOT T0651  ; 入盘机械手前后伺服没归零延时报警
OUT W68.01  ; 入盘机械手前后伺服没归零
TIMX(550) 0651 &120  ; 入盘机械手前后伺服没归零延时报警
; rung 65: 手动报警*****升降伺服
LD W60.01  ; 入盘（升降）Z轴手动下降
OR W60.02  ; 入盘（升降）Z轴手动上升
OR W60.03  ; （龙门）抓料机械手手动取料位置
OR W60.04  ; 入盘（升降）Z轴手动回下料位置
OR W60.05  ; 升降回位
AND A326.05  ; 入盘升降原点标志
OR W68.02  ; 入盘机械手升降伺服没归零
ANDNOT T0652  ; 入盘机械手升降伺服没归零延时报警
OUT W68.02  ; 入盘机械手升降伺服没归零
TIMX(550) 0652 &120  ; 入盘机械手升降伺服没归零延时报警
; rung 66
LDNOT W107.00  ; 入盘（前后）Y轴取料位置
ORNOT W108.15  ; 入盘（左右）X轴左右取料位
@AND W61.00  ; 入盘升降气缸
OR W68.03  ; 入盘升降气缸只能在取料位升降
ANDNOT T0653  ; 入盘升降气缸只能在取料位升降延时
OUT W68.03  ; 入盘升降气缸只能在取料位升降
TIMX(550) 0653 &120  ; 入盘升降气缸只能在取料位升降延时

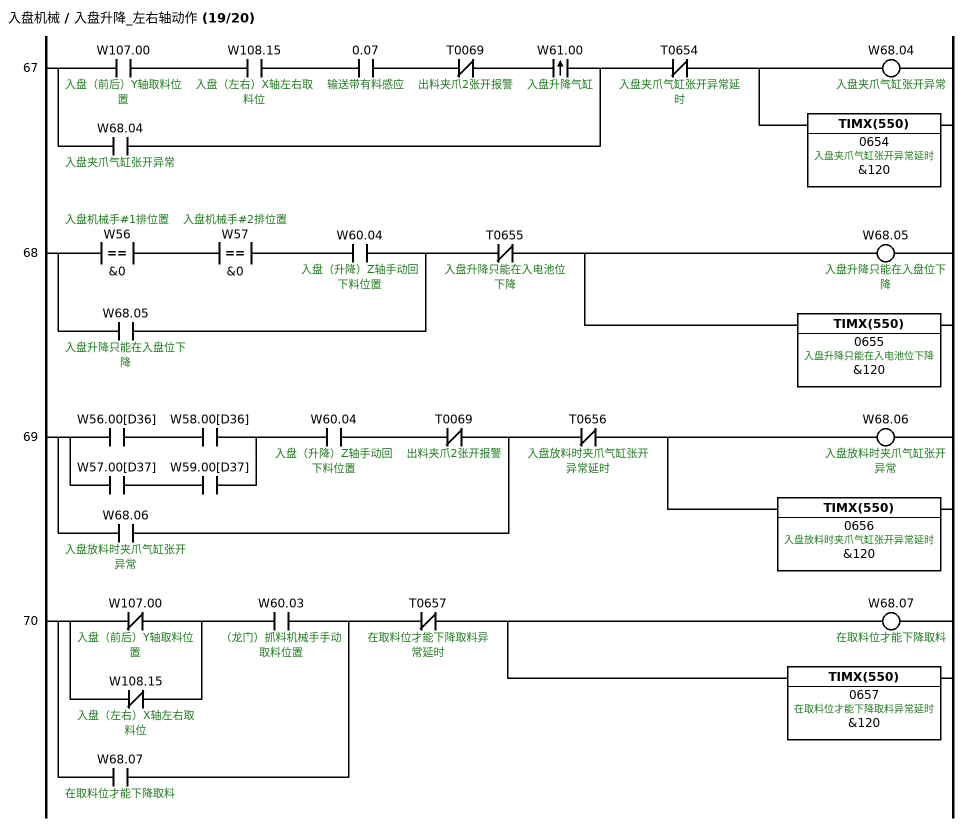
; rung 67
LD W107.00  ; 入盘（前后）Y轴取料位置
AND W108.15  ; 入盘（左右）X轴左右取料位
AND 0.07  ; 输送带有料感应
ANDNOT T0069  ; 出料夹爪2张开报警
@AND W61.00  ; 入盘升降气缸
OR W68.04  ; 入盘夹爪气缸张开异常
ANDNOT T0654  ; 入盘夹爪气缸张开异常延时
OUT W68.04  ; 入盘夹爪气缸张开异常
TIMX(550) 0654 &120  ; 入盘夹爪气缸张开异常延时
; rung 68
LD=(300) W56 &0  ; 入盘机械手#1排位置
AND=(300) W57 &0  ; 入盘机械手#2排位置
AND W60.04  ; 入盘（升降）Z轴手动回下料位置
OR W68.05  ; 入盘升降只能在入盘位下降
ANDNOT T0655  ; 入盘升降只能在入电池位下降
OUT W68.05  ; 入盘升降只能在入盘位下降
TIMX(550) 0655 &120  ; 入盘升降只能在入电池位下降
; rung 69
LD W56.00[D36]
AND W58.00[D36]
LD W57.00[D37]
AND W59.00[D37]
ORLD
AND W60.04  ; 入盘（升降）Z轴手动回下料位置
ANDNOT T0069  ; 出料夹爪2张开报警
OR W68.06  ; 入盘放料时夹爪气缸张开异常
ANDNOT T0656  ; 入盘放料时夹爪气缸张开异常延时
OUT W68.06  ; 入盘放料时夹爪气缸张开异常
TIMX(550) 0656 &120  ; 入盘放料时夹爪气缸张开异常延时
; rung 70
LDNOT W107.00  ; 入盘（前后）Y轴取料位置
ORNOT W108.15  ; 入盘（左右）X轴左右取料位
AND W60.03  ; （龙门）抓料机械手手动取料位置
OR W68.07  ; 在取料位才能下降取料
ANDNOT T0657  ; 在取料位才能下降取料异常延时
OUT W68.07  ; 在取料位才能下降取料
TIMX(550) 0657 &120  ; 在取料位才能下降取料异常延时

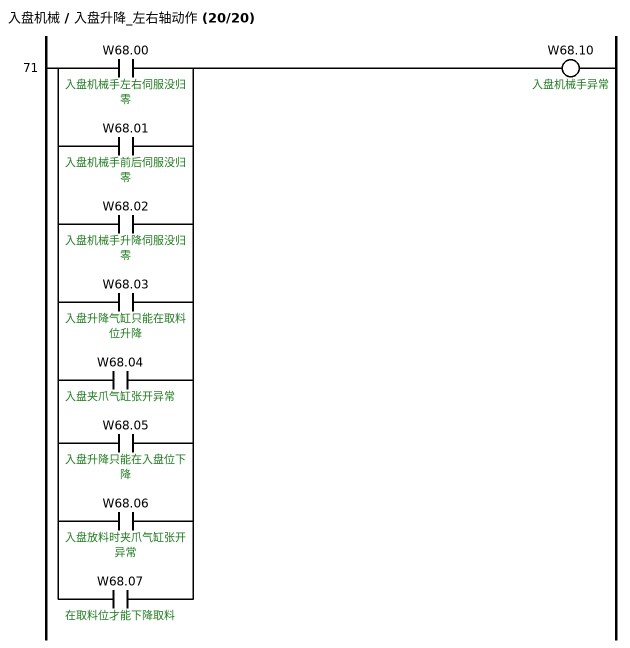
; rung 71
LD W68.00  ; 入盘机械手左右伺服没归零
OR W68.01  ; 入盘机械手前后伺服没归零
OR W68.02  ; 入盘机械手升降伺服没归零
OR W68.03  ; 入盘升降气缸只能在取料位升降
OR W68.04  ; 入盘夹爪气缸张开异常
OR W68.05  ; 入盘升降只能在入盘位下降
OR W68.06  ; 入盘放料时夹爪气缸张开异常
OR W68.07  ; 在取料位才能下降取料
OUT W68.10  ; 入盘机械手异常

### Section 料盒伺服_气缸手动

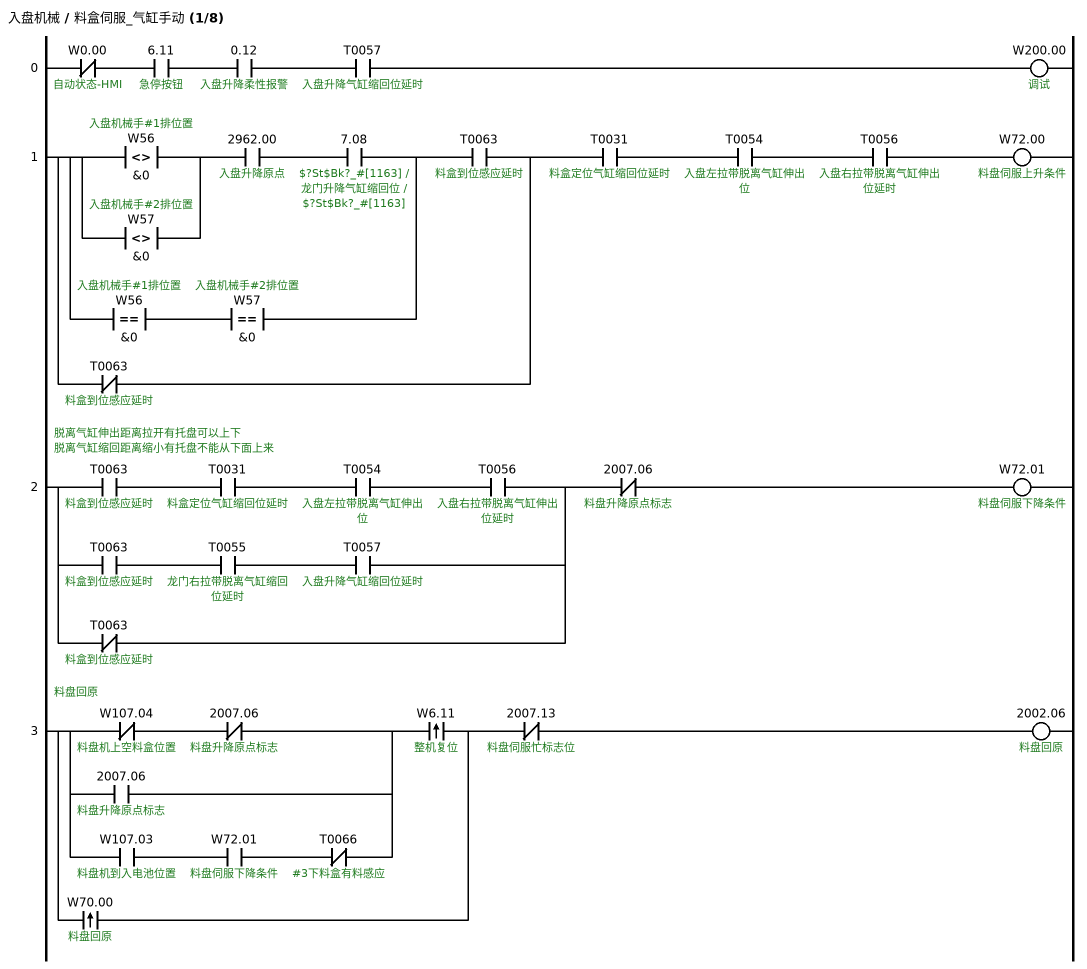
; rung 0
LDNOT W0.00  ; 自动状态-HMI
AND 6.11  ; 急停按钮
AND 0.12  ; 入盘升降柔性报警
AND T0057  ; 入盘升降气缸缩回位延时
OUT W200.00  ; 调试
; rung 1
LD<>(305) W56 &0  ; 入盘机械手#1排位置
OR<>(305) W57 &0  ; 入盘机械手#2排位置
AND 2962.00  ; 入盘升降原点
AND 7.08  ; $?St$Bk?_#[1163] / 龙门升降气缸缩回位 / $?St$Bk?_#[1163]
LD=(300) W56 &0  ; 入盘机械手#1排位置
AND=(300) W57 &0  ; 入盘机械手#2排位置
ORLD
AND T0063  ; 料盒到位感应延时
ORNOT T0063  ; 料盒到位感应延时
AND T0031  ; 料盒定位气缸缩回位延时
AND T0054  ; 入盘左拉带脱离气缸伸出位
AND T0056  ; 入盘右拉带脱离气缸伸出位延时
OUT W72.00  ; 料盘伺服上升条件
; rung 2: 脱离气缸伸出距离拉开有托盘可以上下 / 脱离气缸缩回距离缩小有托盘不能从下面上来
LD T0063  ; 料盒到位感应延时
AND T0031  ; 料盒定位气缸缩回位延时
AND T0054  ; 入盘左拉带脱离气缸伸出位
AND T0056  ; 入盘右拉带脱离气缸伸出位延时
LD T0063  ; 料盒到位感应延时
AND T0055  ; 龙门右拉带脱离气缸缩回位延时
AND T0057  ; 入盘升降气缸缩回位延时
ORLD
ORNOT T0063  ; 料盒到位感应延时
ANDNOT 2007.06  ; 料盘升降原点标志
OUT W72.01  ; 料盘伺服下降条件
; rung 3: 料盘回原
LDNOT W107.04  ; 料盘机上空料盒位置
ANDNOT 2007.06  ; 料盘升降原点标志
OR 2007.06  ; 料盘升降原点标志
LD W107.03  ; 料盘机到入电池位置
AND W72.01  ; 料盘伺服下降条件
ANDNOT T0066  ; #3下料盒有料感应
ORLD
@AND W6.11  ; 整机复位
@OR W70.00  ; 料盘回原
ANDNOT 2007.13  ; 料盘伺服忙标志位
OUT 2002.06  ; 料盘回原

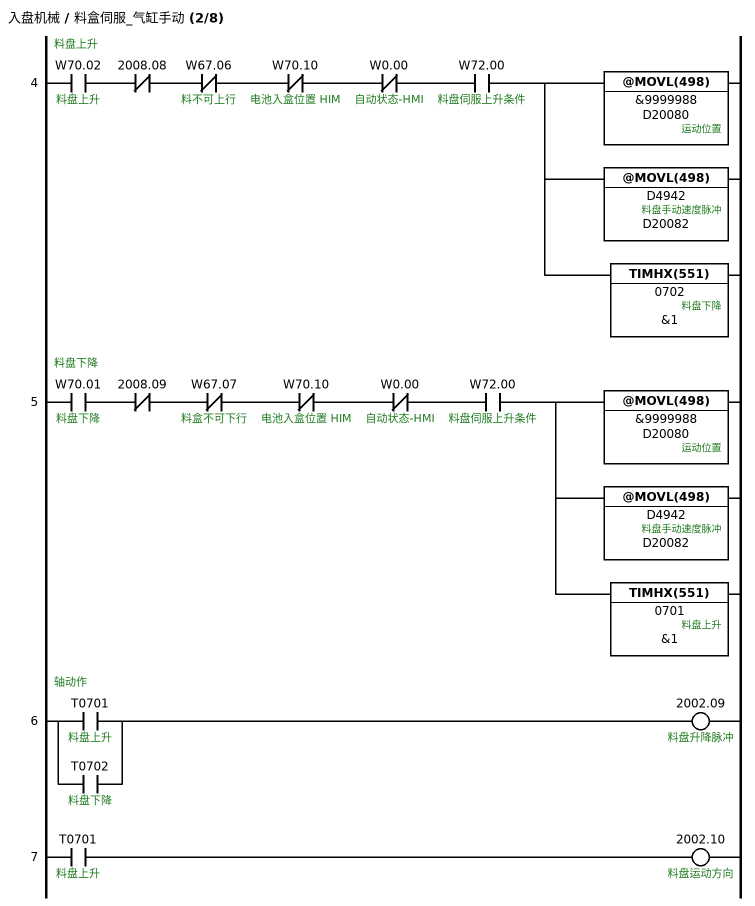
; rung 4: 料盘上升
LD W70.02  ; 料盘上升
ANDNOT 2008.08
ANDNOT W67.06  ; 料不可上行
ANDNOT W70.10  ; 电池入盒位置 HIM
ANDNOT W0.00  ; 自动状态-HMI
AND W72.00  ; 料盘伺服上升条件
@MOVL(498) &9999988 D20080  ; 运动位置
@MOVL(498) D4942 D20082  ; 料盘手动速度脉冲
TIMHX(551) 0702 &1  ; 料盘下降
; rung 5: 料盘下降
LD W70.01  ; 料盘下降
ANDNOT 2008.09
ANDNOT W67.07  ; 料盒不可下行
ANDNOT W70.10  ; 电池入盒位置 HIM
ANDNOT W0.00  ; 自动状态-HMI
AND W72.00  ; 料盘伺服上升条件
@MOVL(498) &9999988 D20080  ; 运动位置
@MOVL(498) D4942 D20082  ; 料盘手动速度脉冲
TIMHX(551) 0701 &1  ; 料盘上升
; rung 6: 轴动作
LD T0701  ; 料盘上升
OR T0702  ; 料盘下降
OUT 2002.09  ; 料盘升降脉冲
; rung 7
LD T0701  ; 料盘上升
OUT 2002.10  ; 料盘运动方向

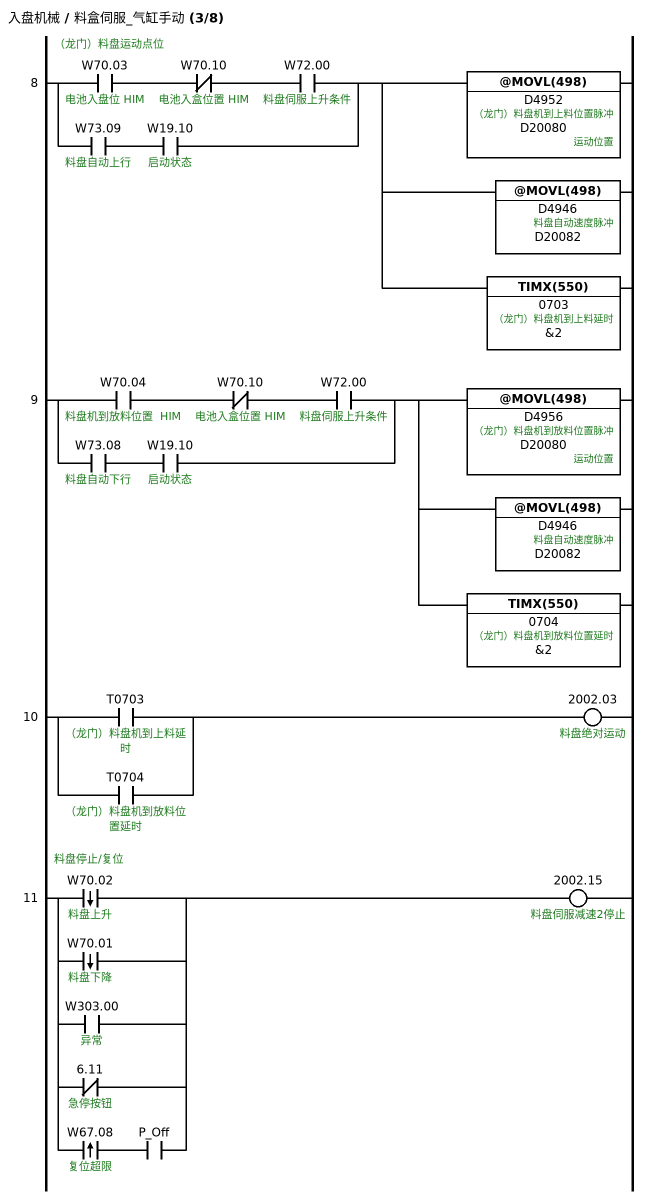
; rung 8: （龙门）料盘运动点位
LD W70.03  ; 电池入盘位 HIM
ANDNOT W70.10  ; 电池入盒位置 HIM
AND W72.00  ; 料盘伺服上升条件
LD W73.09  ; 料盘自动上行
AND W19.10  ; 启动状态
ORLD
@MOVL(498) D4952 D20080  ; （龙门）料盘机到上料位置脉冲, 运动位置
@MOVL(498) D4946 D20082  ; 料盘自动速度脉冲
TIMX(550) 0703 &2  ; （龙门）料盘机到上料延时
; rung 9
LD W70.04  ; 料盘机到放料位置  HIM
ANDNOT W70.10  ; 电池入盒位置 HIM
AND W72.00  ; 料盘伺服上升条件
LD W73.08  ; 料盘自动下行
AND W19.10  ; 启动状态
ORLD
@MOVL(498) D4956 D20080  ; （龙门）料盘机到放料位置脉冲, 运动位置
@MOVL(498) D4946 D20082  ; 料盘自动速度脉冲
TIMX(550) 0704 &2  ; （龙门）料盘机到放料位置延时
; rung 10
LD T0703  ; （龙门）料盘机到上料延时
OR T0704  ; （龙门）料盘机到放料位置延时
OUT 2002.03  ; 料盘绝对运动
; rung 11: 料盘停止/复位
%LD W70.02  ; 料盘上升
%OR W70.01  ; 料盘下降
OR W303.00  ; 异常
ORNOT 6.11  ; 急停按钮
@LD W67.08  ; 复位超限
AND P_Off
ORLD
OUT 2002.15  ; 料盘伺服减速2停止

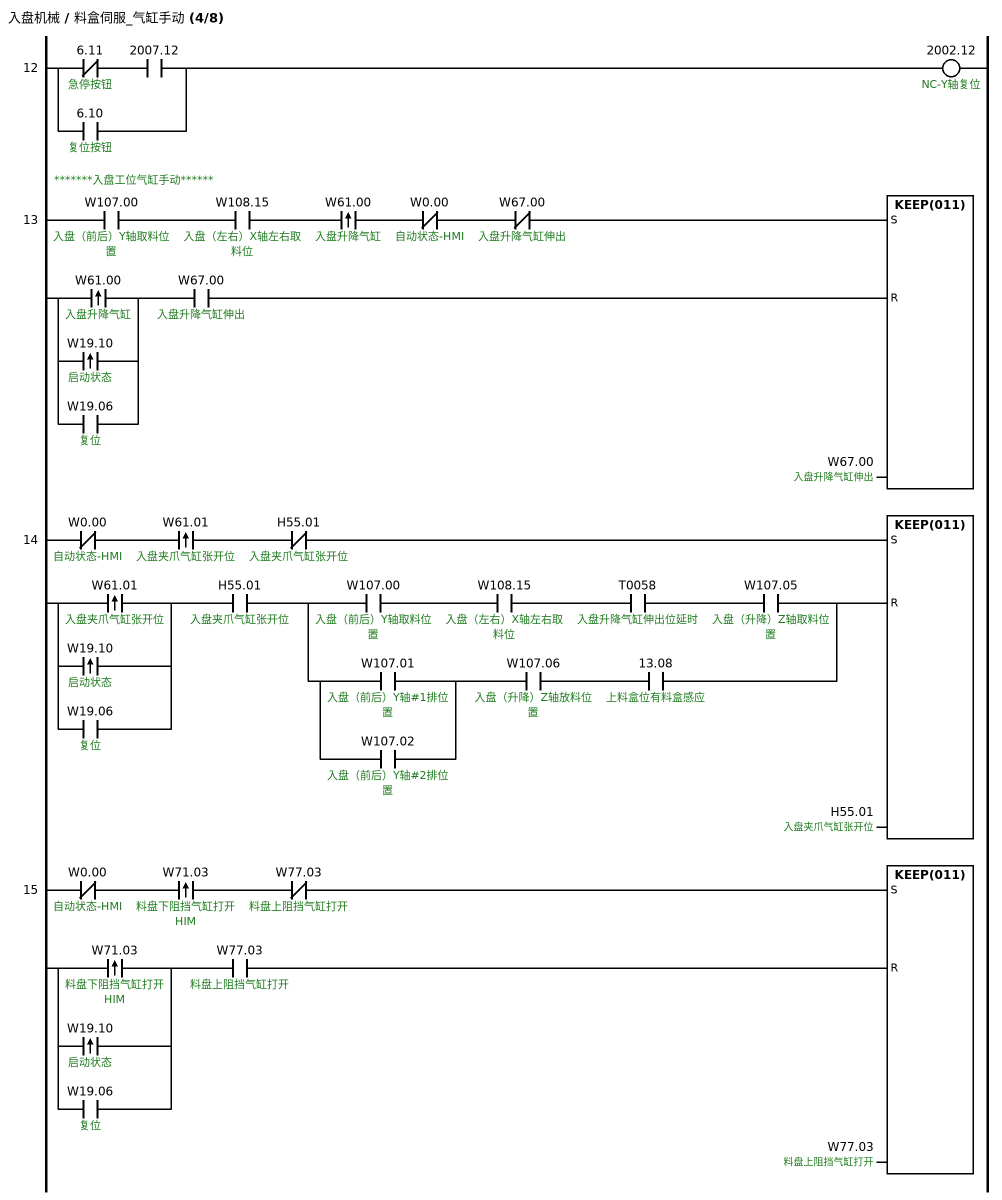
; rung 12
LDNOT 6.11  ; 急停按钮
AND 2007.12
OR 6.10  ; 复位按钮
OUT 2002.12  ; NC-Y轴复位
; rung 13: *******入盘工位气缸手动******
LD W107.00  ; 入盘（前后）Y轴取料位置
AND W108.15  ; 入盘（左右）X轴左右取料位
@AND W61.00  ; 入盘升降气缸
ANDNOT W0.00  ; 自动状态-HMI
ANDNOT W67.00  ; 入盘升降气缸伸出
@LD W61.00  ; 入盘升降气缸
@OR W19.10  ; 启动状态
OR W19.06  ; 复位
AND W67.00  ; 入盘升降气缸伸出
KEEP(011) W67.00  ; 入盘升降气缸伸出
; rung 14
LDNOT W0.00  ; 自动状态-HMI
@AND W61.01  ; 入盘夹爪气缸张开位
ANDNOT H55.01  ; 入盘夹爪气缸张开位
@LD W61.01  ; 入盘夹爪气缸张开位
@OR W19.10  ; 启动状态
OR W19.06  ; 复位
AND H55.01  ; 入盘夹爪气缸张开位
LD W107.00  ; 入盘（前后）Y轴取料位置
AND W108.15  ; 入盘（左右）X轴左右取料位
AND T0058  ; 入盘升降气缸伸出位延时
AND W107.05  ; 入盘（升降）Z轴取料位置
LD W107.01  ; 入盘（前后）Y轴#1排位置
OR W107.02  ; 入盘（前后）Y轴#2排位置
AND W107.06  ; 入盘（升降）Z轴放料位置
AND 13.08  ; 上料盒位有料盒感应
ORLD
ANDLD
KEEP(011) H55.01  ; 入盘夹爪气缸张开位
; rung 15
LDNOT W0.00  ; 自动状态-HMI
@AND W71.03  ; 料盘下阻挡气缸打开  HIM
ANDNOT W77.03  ; 料盘上阻挡气缸打开
@LD W71.03  ; 料盘下阻挡气缸打开  HIM
@OR W19.10  ; 启动状态
OR W19.06  ; 复位
AND W77.03  ; 料盘上阻挡气缸打开
KEEP(011) W77.03  ; 料盘上阻挡气缸打开

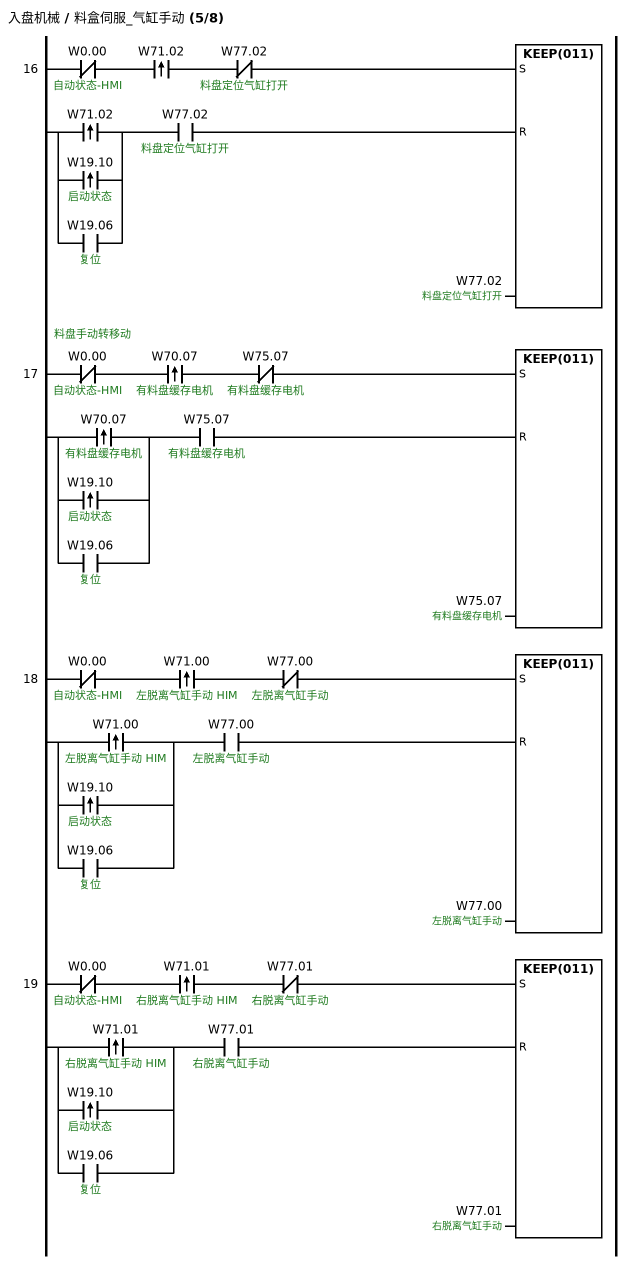
; rung 16
LDNOT W0.00  ; 自动状态-HMI
@AND W71.02
ANDNOT W77.02  ; 料盘定位气缸打开
@LD W71.02
@OR W19.10  ; 启动状态
OR W19.06  ; 复位
AND W77.02  ; 料盘定位气缸打开
KEEP(011) W77.02  ; 料盘定位气缸打开
; rung 17: 料盘手动转移动
LDNOT W0.00  ; 自动状态-HMI
@AND W70.07  ; 有料盘缓存电机
ANDNOT W75.07  ; 有料盘缓存电机
@LD W70.07  ; 有料盘缓存电机
@OR W19.10  ; 启动状态
OR W19.06  ; 复位
AND W75.07  ; 有料盘缓存电机
KEEP(011) W75.07  ; 有料盘缓存电机
; rung 18
LDNOT W0.00  ; 自动状态-HMI
@AND W71.00  ; 左脱离气缸手动 HIM
ANDNOT W77.00  ; 左脱离气缸手动
@LD W71.00  ; 左脱离气缸手动 HIM
@OR W19.10  ; 启动状态
OR W19.06  ; 复位
AND W77.00  ; 左脱离气缸手动
KEEP(011) W77.00  ; 左脱离气缸手动
; rung 19
LDNOT W0.00  ; 自动状态-HMI
@AND W71.01  ; 右脱离气缸手动 HIM
ANDNOT W77.01  ; 右脱离气缸手动
@LD W71.01  ; 右脱离气缸手动 HIM
@OR W19.10  ; 启动状态
OR W19.06  ; 复位
AND W77.01  ; 右脱离气缸手动
KEEP(011) W77.01  ; 右脱离气缸手动

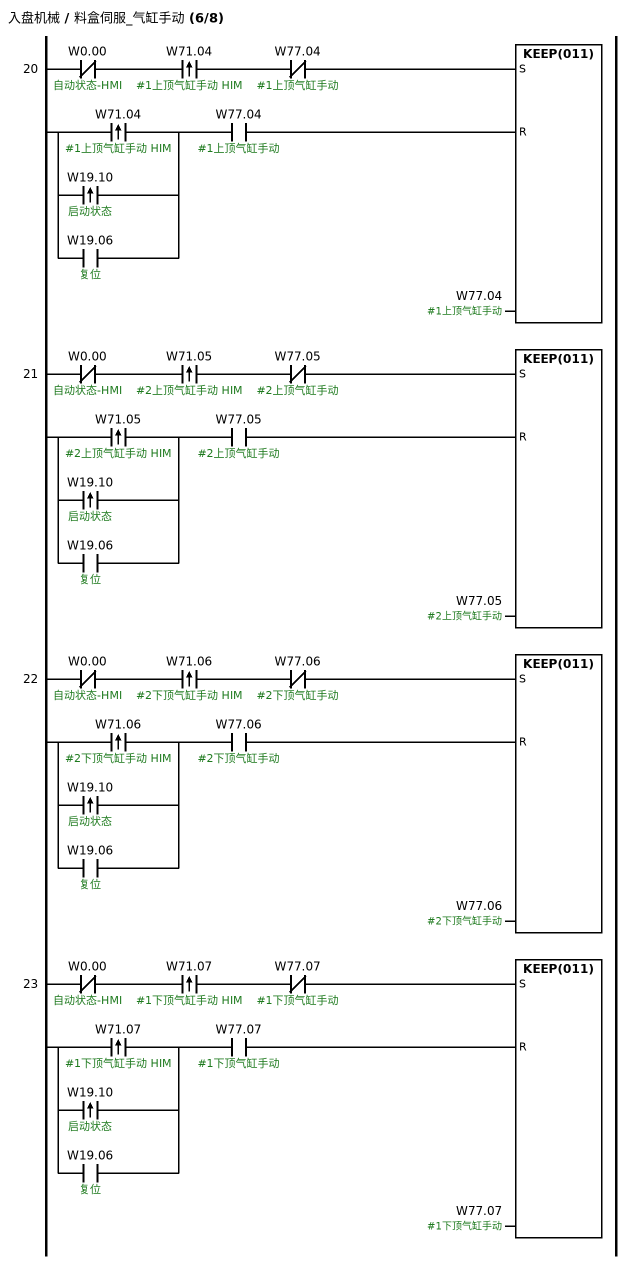
; rung 20
LDNOT W0.00  ; 自动状态-HMI
@AND W71.04  ; #1上顶气缸手动 HIM
ANDNOT W77.04  ; #1上顶气缸手动
@LD W71.04  ; #1上顶气缸手动 HIM
@OR W19.10  ; 启动状态
OR W19.06  ; 复位
AND W77.04  ; #1上顶气缸手动
KEEP(011) W77.04  ; #1上顶气缸手动
; rung 21
LDNOT W0.00  ; 自动状态-HMI
@AND W71.05  ; #2上顶气缸手动 HIM
ANDNOT W77.05  ; #2上顶气缸手动
@LD W71.05  ; #2上顶气缸手动 HIM
@OR W19.10  ; 启动状态
OR W19.06  ; 复位
AND W77.05  ; #2上顶气缸手动
KEEP(011) W77.05  ; #2上顶气缸手动
; rung 22
LDNOT W0.00  ; 自动状态-HMI
@AND W71.06  ; #2下顶气缸手动 HIM
ANDNOT W77.06  ; #2下顶气缸手动
@LD W71.06  ; #2下顶气缸手动 HIM
@OR W19.10  ; 启动状态
OR W19.06  ; 复位
AND W77.06  ; #2下顶气缸手动
KEEP(011) W77.06  ; #2下顶气缸手动
; rung 23
LDNOT W0.00  ; 自动状态-HMI
@AND W71.07  ; #1下顶气缸手动 HIM
ANDNOT W77.07  ; #1下顶气缸手动
@LD W71.07  ; #1下顶气缸手动 HIM
@OR W19.10  ; 启动状态
OR W19.06  ; 复位
AND W77.07  ; #1下顶气缸手动
KEEP(011) W77.07  ; #1下顶气缸手动

